Staubli VAL3: restartMotion.pgx

public program restartMotion()
begin
  // restart the motion
  wait(cycleStatus:bStop==true and cycleStatus:bMoveStopped==true and esStatus()!=2)
  logMsg("[KERNEL] CYCLE:Restart the motion")
  // reset the bit
  cycleStatus:bStop=false
end
